// TIA Portal V16 export
// export: Created 2024-09-05T17:39:08.8443912Z, ExportSetting WithDefaults, DisplayName Totally Integrated Automation Portal, DisplayVersion V16 Update 6, DisplayName TIA Portal Version Control Interface, DisplayVersion V16 Update 2, DisplayName TIA Portal Openness, DisplayVersion V16 Update 6, DisplayName STEP 7 Professional, DisplayVersion V16 Update 6, DisplayName STEP 7 Safety, DisplayVersion V16, DisplayName WinCC Advanced, DisplayVersion V16 Update 6
DATA_BLOCK "DigiforceMain_DB"   // DB47
VERSION : 0.1
// stored: AutoNumber true, DBAccessibleFromOPCUA true, InstanceOfName DigiforceMain, InstanceOfType FB
"DigiforceMain"
   // VAR
   //    Digiforce1_Instance { S7_SetPoint := 'True'} : "Digiforce";
   //    Digiforce2_Instance { S7_SetPoint := 'True'} : "Digiforce";
   //    Digiforce3_Instance { S7_SetPoint := 'True'} : "Digiforce";
   //    Digiforce4_Instance { S7_SetPoint := 'True'} : "Digiforce";
   // END_VAR
BEGIN
   Digiforce1_Instance.DataRead := 488;
   Digiforce1_Instance.DataWrite := 487;
   Digiforce1_Instance.send.Tare_X := FALSE;
   Digiforce1_Instance.send.Res_Stat := FALSE;
   Digiforce1_Instance.send.Stest := FALSE;
   Digiforce1_Instance.send.Strobe := FALSE;
   Digiforce1_Instance.send.Auto := FALSE;
   Digiforce1_Instance.send.reserve1 := FALSE;
   Digiforce1_Instance.send.reserve2 := FALSE;
   Digiforce1_Instance.send.reserve3 := FALSE;
   Digiforce1_Instance.send.Prog := 16#00;
   Digiforce1_Instance.send.Start := FALSE;
   Digiforce1_Instance.receive.dataD.Ready := TRUE;
   Digiforce1_Instance.receive.dataD.OK := FALSE;
   Digiforce1_Instance.receive.dataD.NOK := TRUE;
   Digiforce1_Instance.receive.dataD.NOK_ONL := FALSE;
   Digiforce1_Instance.receive.dataD.S1 := TRUE;
   Digiforce1_Instance.receive.dataD.S2 := FALSE;
   Digiforce1_Instance.receive.dataD.OK_STEST := FALSE;
   Digiforce1_Instance.receive.dataD.MEAS_ACT := FALSE;
   Digiforce1_Instance.receive.dataD.Strobe := FALSE;
   Digiforce1_Instance.receive.dataD.Prog0 := FALSE;
   Digiforce1_Instance.receive.dataD.Prog1 := FALSE;
   Digiforce1_Instance.receive.dataD.Prog2 := FALSE;
   Digiforce1_Instance.receive.dataD.reserve1 := FALSE;
   Digiforce1_Instance.receive.dataD.reserve2 := FALSE;
   Digiforce1_Instance.receive.dataD.reserve3 := FALSE;
   Digiforce1_Instance.receive.dataD.reserve4 := FALSE;
   Digiforce1_Instance.receive.dataD.Global_NOK := TRUE;
   Digiforce1_Instance.receive.dataD."Overload _NOK" := FALSE;
   Digiforce1_Instance.receive.dataD.Window_1_NOK := TRUE;
   Digiforce1_Instance.receive.dataD.Window_2_NOK := FALSE;
   Digiforce1_Instance.receive.dataD.Window_3_NOK := FALSE;
   Digiforce1_Instance.receive.dataD.Threshold_1_NOK := TRUE;
   Digiforce1_Instance.receive.dataD.Threshold_2_NOK := FALSE;
   Digiforce1_Instance.receive.dataD.Trapezoid_1_NOK := FALSE;
   Digiforce1_Instance.receive.dataD.Trapezoid2_NOK := FALSE;
   Digiforce1_Instance.receive.dataD.Envelope_NOK := FALSE;
   Digiforce1_Instance.receive.dataD."Measurement_w/o_READY" := FALSE;
   Digiforce1_Instance.receive.dataD.USB_logging_error := FALSE;
   Digiforce1_Instance.receive.dataD.reserve5 := FALSE;
   Digiforce1_Instance.receive.dataD.reserve6 := FALSE;
   Digiforce1_Instance.receive.dataD.reserve7 := FALSE;
   Digiforce1_Instance.receive.dataD.reserve8 := FALSE;
   Digiforce1_Instance.receive.dataA[1..20] := 909090.0;
   Digiforce1_Instance.receive.dataA[21] := 8.063384;
   Digiforce1_Instance.receive.dataA[22] := -0.03242895;
   Digiforce1_Instance.IEC_Timer_zmenaProgramu.PT := T#0MS;
   Digiforce1_Instance.IEC_Timer_zmenaProgramu.IN := FALSE;
   Digiforce2_Instance.DataRead := 548;
   Digiforce2_Instance.DataWrite := 547;
   Digiforce2_Instance.send.Tare_X := FALSE;
   Digiforce2_Instance.send.Res_Stat := FALSE;
   Digiforce2_Instance.send.Stest := FALSE;
   Digiforce2_Instance.send.Strobe := FALSE;
   Digiforce2_Instance.send.Auto := FALSE;
   Digiforce2_Instance.send.reserve1 := FALSE;
   Digiforce2_Instance.send.reserve2 := FALSE;
   Digiforce2_Instance.send.reserve3 := FALSE;
   Digiforce2_Instance.send.Prog := 16#00;
   Digiforce2_Instance.send.Start := FALSE;
   Digiforce2_Instance.receive.dataD.Ready := TRUE;
   Digiforce2_Instance.receive.dataD.OK := FALSE;
   Digiforce2_Instance.receive.dataD.NOK := TRUE;
   Digiforce2_Instance.receive.dataD.NOK_ONL := FALSE;
   Digiforce2_Instance.receive.dataD.S1 := TRUE;
   Digiforce2_Instance.receive.dataD.S2 := FALSE;
   Digiforce2_Instance.receive.dataD.OK_STEST := FALSE;
   Digiforce2_Instance.receive.dataD.MEAS_ACT := FALSE;
   Digiforce2_Instance.receive.dataD.Strobe := FALSE;
   Digiforce2_Instance.receive.dataD.Prog0 := FALSE;
   Digiforce2_Instance.receive.dataD.Prog1 := FALSE;
   Digiforce2_Instance.receive.dataD.Prog2 := FALSE;
   Digiforce2_Instance.receive.dataD.reserve1 := FALSE;
   Digiforce2_Instance.receive.dataD.reserve2 := FALSE;
   Digiforce2_Instance.receive.dataD.reserve3 := FALSE;
   Digiforce2_Instance.receive.dataD.reserve4 := FALSE;
   Digiforce2_Instance.receive.dataD.Global_NOK := TRUE;
   Digiforce2_Instance.receive.dataD."Overload _NOK" := FALSE;
   Digiforce2_Instance.receive.dataD.Window_1_NOK := TRUE;
   Digiforce2_Instance.receive.dataD.Window_2_NOK := FALSE;
   Digiforce2_Instance.receive.dataD.Window_3_NOK := FALSE;
   Digiforce2_Instance.receive.dataD.Threshold_1_NOK := TRUE;
   Digiforce2_Instance.receive.dataD.Threshold_2_NOK := FALSE;
   Digiforce2_Instance.receive.dataD.Trapezoid_1_NOK := FALSE;
   Digiforce2_Instance.receive.dataD.Trapezoid2_NOK := FALSE;
   Digiforce2_Instance.receive.dataD.Envelope_NOK := FALSE;
   Digiforce2_Instance.receive.dataD."Measurement_w/o_READY" := FALSE;
   Digiforce2_Instance.receive.dataD.USB_logging_error := FALSE;
   Digiforce2_Instance.receive.dataD.reserve5 := FALSE;
   Digiforce2_Instance.receive.dataD.reserve6 := FALSE;
   Digiforce2_Instance.receive.dataD.reserve7 := FALSE;
   Digiforce2_Instance.receive.dataD.reserve8 := FALSE;
   Digiforce2_Instance.receive.dataA[1..20] := 909090.0;
   Digiforce2_Instance.receive.dataA[21] := 8.028815;
   Digiforce2_Instance.receive.dataA[22] := -0.02130306;
   Digiforce2_Instance.IEC_Timer_zmenaProgramu.PT := T#0MS;
   Digiforce2_Instance.IEC_Timer_zmenaProgramu.IN := FALSE;
   Digiforce3_Instance.DataRead := 610;
   Digiforce3_Instance.DataWrite := 609;
   Digiforce3_Instance.send.Tare_X := FALSE;
   Digiforce3_Instance.send.Res_Stat := FALSE;
   Digiforce3_Instance.send.Stest := FALSE;
   Digiforce3_Instance.send.Strobe := FALSE;
   Digiforce3_Instance.send.Auto := FALSE;
   Digiforce3_Instance.send.reserve1 := FALSE;
   Digiforce3_Instance.send.reserve2 := FALSE;
   Digiforce3_Instance.send.reserve3 := FALSE;
   Digiforce3_Instance.send.Prog := 16#01;
   Digiforce3_Instance.send.Start := FALSE;
   Digiforce3_Instance.receive.dataD.Ready := TRUE;
   Digiforce3_Instance.receive.dataD.OK := FALSE;
   Digiforce3_Instance.receive.dataD.NOK := TRUE;
   Digiforce3_Instance.receive.dataD.NOK_ONL := FALSE;
   Digiforce3_Instance.receive.dataD.S1 := TRUE;
   Digiforce3_Instance.receive.dataD.S2 := FALSE;
   Digiforce3_Instance.receive.dataD.OK_STEST := FALSE;
   Digiforce3_Instance.receive.dataD.MEAS_ACT := FALSE;
   Digiforce3_Instance.receive.dataD.Strobe := FALSE;
   Digiforce3_Instance.receive.dataD.Prog0 := TRUE;
   Digiforce3_Instance.receive.dataD.Prog1 := FALSE;
   Digiforce3_Instance.receive.dataD.Prog2 := FALSE;
   Digiforce3_Instance.receive.dataD.reserve1 := FALSE;
   Digiforce3_Instance.receive.dataD.reserve2 := FALSE;
   Digiforce3_Instance.receive.dataD.reserve3 := FALSE;
   Digiforce3_Instance.receive.dataD.reserve4 := FALSE;
   Digiforce3_Instance.receive.dataD.Global_NOK := TRUE;
   Digiforce3_Instance.receive.dataD."Overload _NOK" := FALSE;
   Digiforce3_Instance.receive.dataD.Window_1_NOK := TRUE;
   Digiforce3_Instance.receive.dataD.Window_2_NOK := FALSE;
   Digiforce3_Instance.receive.dataD.Window_3_NOK := FALSE;
   Digiforce3_Instance.receive.dataD.Threshold_1_NOK := TRUE;
   Digiforce3_Instance.receive.dataD.Threshold_2_NOK := FALSE;
   Digiforce3_Instance.receive.dataD.Trapezoid_1_NOK := FALSE;
   Digiforce3_Instance.receive.dataD.Trapezoid2_NOK := FALSE;
   Digiforce3_Instance.receive.dataD.Envelope_NOK := FALSE;
   Digiforce3_Instance.receive.dataD."Measurement_w/o_READY" := FALSE;
   Digiforce3_Instance.receive.dataD.USB_logging_error := FALSE;
   Digiforce3_Instance.receive.dataD.reserve5 := FALSE;
   Digiforce3_Instance.receive.dataD.reserve6 := FALSE;
   Digiforce3_Instance.receive.dataD.reserve7 := FALSE;
   Digiforce3_Instance.receive.dataD.reserve8 := FALSE;
   Digiforce3_Instance.receive.dataA[1..20] := 909090.0;
   Digiforce3_Instance.receive.dataA[21] := 8.030701;
   Digiforce3_Instance.receive.dataA[22] := -0.01457718;
   Digiforce3_Instance.IEC_Timer_zmenaProgramu.PT := T#10S;
   Digiforce3_Instance.IEC_Timer_zmenaProgramu.IN := FALSE;
   Digiforce4_Instance.DataRead := 672;
   Digiforce4_Instance.DataWrite := 671;
   Digiforce4_Instance.send.Tare_X := FALSE;
   Digiforce4_Instance.send.Res_Stat := FALSE;
   Digiforce4_Instance.send.Stest := FALSE;
   Digiforce4_Instance.send.Strobe := FALSE;
   Digiforce4_Instance.send.Auto := FALSE;
   Digiforce4_Instance.send.reserve1 := FALSE;
   Digiforce4_Instance.send.reserve2 := FALSE;
   Digiforce4_Instance.send.reserve3 := FALSE;
   Digiforce4_Instance.send.Prog := 16#01;
   Digiforce4_Instance.send.Start := FALSE;
   Digiforce4_Instance.receive.dataD.Ready := TRUE;
   Digiforce4_Instance.receive.dataD.OK := FALSE;
   Digiforce4_Instance.receive.dataD.NOK := TRUE;
   Digiforce4_Instance.receive.dataD.NOK_ONL := FALSE;
   Digiforce4_Instance.receive.dataD.S1 := TRUE;
   Digiforce4_Instance.receive.dataD.S2 := FALSE;
   Digiforce4_Instance.receive.dataD.OK_STEST := FALSE;
   Digiforce4_Instance.receive.dataD.MEAS_ACT := FALSE;
   Digiforce4_Instance.receive.dataD.Strobe := FALSE;
   Digiforce4_Instance.receive.dataD.Prog0 := TRUE;
   Digiforce4_Instance.receive.dataD.Prog1 := FALSE;
   Digiforce4_Instance.receive.dataD.Prog2 := FALSE;
   Digiforce4_Instance.receive.dataD.reserve1 := FALSE;
   Digiforce4_Instance.receive.dataD.reserve2 := FALSE;
   Digiforce4_Instance.receive.dataD.reserve3 := FALSE;
   Digiforce4_Instance.receive.dataD.reserve4 := FALSE;
   Digiforce4_Instance.receive.dataD.Global_NOK := TRUE;
   Digiforce4_Instance.receive.dataD."Overload _NOK" := FALSE;
   Digiforce4_Instance.receive.dataD.Window_1_NOK := TRUE;
   Digiforce4_Instance.receive.dataD.Window_2_NOK := FALSE;
   Digiforce4_Instance.receive.dataD.Window_3_NOK := FALSE;
   Digiforce4_Instance.receive.dataD.Threshold_1_NOK := TRUE;
   Digiforce4_Instance.receive.dataD.Threshold_2_NOK := FALSE;
   Digiforce4_Instance.receive.dataD.Trapezoid_1_NOK := FALSE;
   Digiforce4_Instance.receive.dataD.Trapezoid2_NOK := FALSE;
   Digiforce4_Instance.receive.dataD.Envelope_NOK := FALSE;
   Digiforce4_Instance.receive.dataD."Measurement_w/o_READY" := FALSE;
   Digiforce4_Instance.receive.dataD.USB_logging_error := FALSE;
   Digiforce4_Instance.receive.dataD.reserve5 := FALSE;
   Digiforce4_Instance.receive.dataD.reserve6 := FALSE;
   Digiforce4_Instance.receive.dataD.reserve7 := FALSE;
   Digiforce4_Instance.receive.dataD.reserve8 := FALSE;
   Digiforce4_Instance.receive.dataA[1..20] := 909090.0;
   Digiforce4_Instance.receive.dataA[21] := 8.018154;
   Digiforce4_Instance.receive.dataA[22] := -0.01945436;
   Digiforce4_Instance.IEC_Timer_zmenaProgramu.PT := T#10S;
   Digiforce4_Instance.IEC_Timer_zmenaProgramu.IN := FALSE;
END_DATA_BLOCK
